{attribute 'GeneratedUsingTerminal: APS4322-5000-0017'}
{attribute addProperty BoxType "APS4322-5000-0017"}
{attribute addProperty Id "EtcSlaveTerminalBaseFB_InputsAT %I*FB_Inputs_F0F03BDD308WcStateAT %I*WcState_9091E0EB2InfoDataAT %I*InfoData_A7436BC610"}
{attribute addProperty CRC "1955586241"}
{attribute addProperty Size "320"}
TYPE APS4322_748FE0C1 EXTENDS EtcSlaveTerminalBase :
STRUCT
	{attribute addProperty Name "FB_Inputs"}
	FB_Inputs : FB_Inputs_F0F03BDD;
	{attribute addProperty Name "WcState"}
	WcState : WcState_9091E0EB;
	{attribute addProperty Name "InfoData"}
	InfoData : InfoData_A7436BC6;
END_STRUCT
END_TYPE

(* stored: Version 1.2.0.0, ProductVersion 3.1.4024.9
   DUT APS4322_748FE0C1: Id {a5948aea-dffa-4a89-827b-dbad9b8ccbdc} *)
